# EPICS autosave request: photronApp/Db/Photron_settings.req
file "ADBase_settings.req", P=$(P), R=$(R)

#
$(P)$(R)8BitSel
